// TIA Portal V19 export
TYPE "LEXCHANGETRAY_typeTrayInterface"
// stored: Access Published
   STRUCT
      monitor { S7_SetPoint := 'True'} : "LEXCHANGETRAY_typeTrayMonitor";
      commands { S7_SetPoint := 'True'} : "LEXCHANGETRAY_typeTrayCommands";
   END_STRUCT;
END_TYPE
